// TIA Portal V15.1 export
// export: Created 2024-05-17T05:38:32.8666794Z, ExportSetting WithDefaults, DisplayName Totally Integrated Automation Portal, DisplayVersion V15.1 Update 5, DisplayName TIA Portal Openness, DisplayVersion V15.1 Update 5, DisplayName SINAMICS Startdrive Advanced, DisplayVersion V15.1, DisplayName G130, G150, S120, S150, SINAMICS MV, S210, DisplayVersion V15.1, DisplayName G110M, G120, G120C, G120D, G120P, DisplayVersion V15.1, DisplayName STEP 7 Professional, DisplayVersion V15.1 Update 5, DisplayName STEP 7 Safety, DisplayVersion V15.1, DisplayName WinCC Professional, DisplayVersion V15.1 Update 5, DisplayName SIMATIC Visualization Architect, DisplayVersion V15.1
FUNCTION_BLOCK "LAnInput2Lim"   // FB1707, FBD
TITLE = LAnInput2Lim
{ S7_Optimized_Access := 'FALSE' }
AUTHOR : VCC
FAMILY : ProcEqp
NAME : AnInput2
VERSION : 1.0
// ================================================================================
// This module is used to read an analogue Input value and scale it. 
// It also gives the possibility to define 2 limits (High and Low) and to create  
// alarms for these limits. 
// ================================================================================
// stored: AutoNumber false, IsIECCheckEnabled false, SetENOAutomatically False, UDAEnableTagReadback false
   VAR_INPUT
      I_AnInput { ExternalAccessible := 'False'; ExternalVisible := 'False'; ExternalWritable := 'False'} : Int;   // Analogue Input Value
      I_AnInput_Bipolar { ExternalAccessible := 'False'; ExternalVisible := 'False'; ExternalWritable := 'False'} : Bool;   // TRUE if Analogue Input Bipolar
      I_EnHAlarm { ExternalAccessible := 'False'; ExternalVisible := 'False'; ExternalWritable := 'False'} : Bool;   // Enable H Limit Alarm
      I_ResHAlarm { ExternalAccessible := 'False'; ExternalVisible := 'False'; ExternalWritable := 'False'} : Bool;   // Reset H Limit Alarm
      I_EnLAlarm { ExternalAccessible := 'False'; ExternalVisible := 'False'; ExternalWritable := 'False'} : Bool;   // Enable L Limit Alarm
      I_ResLAlarm { ExternalAccessible := 'False'; ExternalVisible := 'False'; ExternalWritable := 'False'} : Bool;   // Reset L Limit Alarm
      I_AlarmResetPB { ExternalAccessible := 'False'; ExternalVisible := 'False'; ExternalWritable := 'False'} : Bool;   // Alarm reset PB
   END_VAR
   VAR_OUTPUT
      O_SensorAlarm { ExternalAccessible := 'False'; ExternalVisible := 'False'; ExternalWritable := 'False'} : Bool;   // Sensor out of range
      O_HAlarm { ExternalAccessible := 'False'; ExternalVisible := 'False'; ExternalWritable := 'False'} : Bool;   // H Limit Alarm
      O_LAlarm { ExternalAccessible := 'False'; ExternalVisible := 'False'; ExternalWritable := 'False'} : Bool;   // L Limit Alarm
      O_AnInputScaled : Real;   // Analogue Input value after scaling
      O_AlarmABCondition { ExternalAccessible := 'False'; ExternalVisible := 'False'; ExternalWritable := 'False'} : Bool;   // Alarm AB condition
      O_HReached { ExternalAccessible := 'False'; ExternalVisible := 'False'; ExternalWritable := 'False'} : Bool;   // High Limit Reached
      O_LReached { ExternalAccessible := 'False'; ExternalVisible := 'False'; ExternalWritable := 'False'} : Bool;   // Low Limit Reached
      H_IAnim { ExternalAccessible := 'False'; ExternalVisible := 'False'; ExternalWritable := 'False'} : Word;   // HMI Animation of the icon
   END_VAR
   VAR DB_SPECIFIC
      H_In : Struct   // HMI
         AnInput_HighLimit : Real;   // From HMI : High Limit For Scaling Analogue Input
         AnInput_LowLimit : Real;   // From HMI : Low Limit For Scaling Analogue Input
         HHysteresis : Real;   // From HMI : Hysteresis value for High Limits
         LHysteresis : Real;   // From HMI : Hysteresis value for Low Limits
         HLimitValue : Real;   // From HMI : High Limit Value
         LLimitValue : Real;   // From HMI : Low Limit Value
         TimeDelay : DInt;   // From HMI : Time delay for limits
         Forcing : Bool;   // From HMI : True if forced value must be used
         ForcedAnInput : Real;   // From HMI : Forced Analogue Input Value
      END_STRUCT;
      H_Out : Struct   // HMI
         Anim : Word;   // HMI Animation of the object
         DBnr : Int;   // HMI Animation DB number
      END_STRUCT;
   END_VAR
   VAR
      HLimitTimer { ExternalAccessible := 'False'; ExternalVisible := 'False'; ExternalWritable := 'False'; S7_SetPoint := 'True'} : "LTimer";   // Timer H Limit
      LLimitTimer { ExternalAccessible := 'False'; ExternalVisible := 'False'; ExternalWritable := 'False'; S7_SetPoint := 'True'} : "LTimer";   // Timer L Limit
   END_VAR
   VAR DB_SPECIFIC
      AnInputScaled { ExternalAccessible := 'False'; ExternalVisible := 'False'; ExternalWritable := 'False'} : Real;   // Analogue Input value after scaling
      HTempSR { ExternalAccessible := 'False'; ExternalVisible := 'False'; ExternalWritable := 'False'} : Bool;   // Temp variable for SET/RESET
      LTempSR { ExternalAccessible := 'False'; ExternalVisible := 'False'; ExternalWritable := 'False'} : Bool;   // Temp variable for SET/RESET
      Scale_status { ExternalAccessible := 'False'; ExternalVisible := 'False'; ExternalWritable := 'False'} : Word;   // Status word for scaling operation
      HlimitHyst { ExternalAccessible := 'False'; ExternalVisible := 'False'; ExternalWritable := 'False'} : Real;   // H Limit with Hysteresis
      LlimitHyst { ExternalAccessible := 'False'; ExternalVisible := 'False'; ExternalWritable := 'False'} : Real;   // L Limit with Hysteresis
      HReached { ExternalAccessible := 'False'; ExternalVisible := 'False'; ExternalWritable := 'False'} : Bool;   // Temp variable H Limit Reached
      LReached { ExternalAccessible := 'False'; ExternalVisible := 'False'; ExternalWritable := 'False'} : Bool;   // Temp variable L Limit Reached
      HAlarmAlmCond { ExternalAccessible := 'False'; ExternalVisible := 'False'; ExternalWritable := 'False'} : Bool;   // HAlarm alarm condition
      LAlarmAlmCond { ExternalAccessible := 'False'; ExternalVisible := 'False'; ExternalWritable := 'False'} : Bool;   // LAlarm alarm condition
      HAlarm { ExternalAccessible := 'False'; ExternalVisible := 'False'; ExternalWritable := 'False'} : Bool;   // H Limit Alarm
      LAlarm { ExternalAccessible := 'False'; ExternalVisible := 'False'; ExternalWritable := 'False'} : Bool;   // L Limit Alarm
      SensorAlarm { ExternalAccessible := 'False'; ExternalVisible := 'False'; ExternalWritable := 'False'} : Bool;   // Sensor out of range
      SensorAlmCond { ExternalAccessible := 'False'; ExternalVisible := 'False'; ExternalWritable := 'False'} : Bool;   // Sensor alarm condition
      ScaleRetValue { ExternalAccessible := 'False'; ExternalVisible := 'False'; ExternalWritable := 'False'} : Int;   // Scale return value
      AnInputTmp { ExternalAccessible := 'False'; ExternalVisible := 'False'; ExternalWritable := 'False'} : Real;   // Analog input temporary
      DBnr { ExternalAccessible := 'False'; ExternalVisible := 'False'; ExternalWritable := 'False'} : Int;   // HMI DB number
   END_VAR
   VAR
      H_Alarm { ExternalAccessible := 'False'; ExternalVisible := 'False'; ExternalWritable := 'False'; S7_SetPoint := 'True'} : "LProc1AlarmMultiIn";
      L_Alarm { ExternalAccessible := 'False'; ExternalVisible := 'False'; ExternalWritable := 'False'; S7_SetPoint := 'True'} : "LProc1AlarmMultiIn";
      SensorAlm { ExternalAccessible := 'False'; ExternalVisible := 'False'; ExternalWritable := 'False'; S7_SetPoint := 'True'} : "LProc1AlarmMultiIn";
   END_VAR
BEGIN

NETWORK
TITLE = **** 1 - Inputs **** DB number
// DB number
      L     DINO;
      T     #DBnr;

REGION Network 2: **** 2.2 - Alarms - Alarm generation **** Alarm High Limit
   // Alarm High Limit
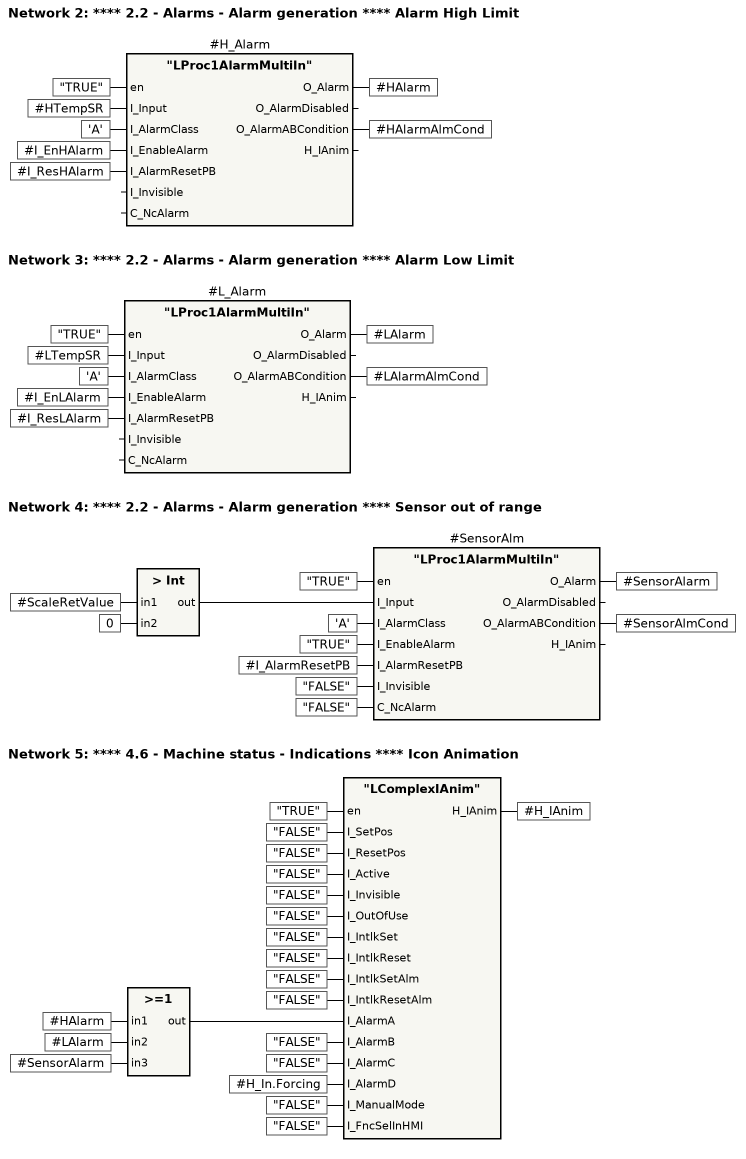
   IF "TRUE" THEN
       #H_Alarm(I_Input := #HTempSR,   // "LProc1AlarmMultiIn"
                I_AlarmClass := 'A',
                I_EnableAlarm := #I_EnHAlarm,
                I_AlarmResetPB := #I_ResHAlarm,
                O_Alarm => #HAlarm,
                O_AlarmABCondition => #HAlarmAlmCond);
   END_IF;
END_REGION

REGION Network 3: **** 2.2 - Alarms - Alarm generation **** Alarm Low Limit
   // Alarm Low Limit
   IF "TRUE" THEN
       #L_Alarm(I_Input := #LTempSR,   // "LProc1AlarmMultiIn"
                I_AlarmClass := 'A',
                I_EnableAlarm := #I_EnLAlarm,
                I_AlarmResetPB := #I_ResLAlarm,
                O_Alarm => #LAlarm,
                O_AlarmABCondition => #LAlarmAlmCond);
   END_IF;
END_REGION

REGION Network 4: **** 2.2 - Alarms - Alarm generation **** Sensor out of range
   // Sensor out of range
   IF "TRUE" THEN
       #SensorAlm(I_Input := #ScaleRetValue > 0,   // "LProc1AlarmMultiIn"
                  I_AlarmClass := 'A',
                  I_EnableAlarm := "TRUE",
                  I_AlarmResetPB := #I_AlarmResetPB,
                  I_Invisible := "FALSE",
                  C_NcAlarm := "FALSE",
                  O_Alarm => #SensorAlarm,
                  O_AlarmABCondition => #SensorAlmCond);
   END_IF;
END_REGION

REGION Network 5: **** 4.6 - Machine status - Indications **** Icon Animation
   // Icon Animation
   IF "TRUE" THEN
       "LComplexIAnim"(I_SetPos := "FALSE",
                       I_ResetPos := "FALSE",
                       I_Active := "FALSE",
                       I_Invisible := "FALSE",
                       I_OutOfUse := "FALSE",
                       I_IntlkSet := "FALSE",
                       I_IntlkReset := "FALSE",
                       I_IntlkSetAlm := "FALSE",
                       I_IntlkResetAlm := "FALSE",
                       I_AlarmA := #HAlarm OR #LAlarm OR #SensorAlarm,
                       I_AlarmB := "FALSE",
                       I_AlarmC := "FALSE",
                       I_AlarmD := #H_In.Forcing,
                       I_ManualMode := "FALSE",
                       I_FncSelInHMI := "FALSE",
                       H_IAnim => #H_IAnim);
   END_IF;
END_REGION

REGION Network 6: **** 4.6 - Machine status - Indications **** Animation
   // Animation
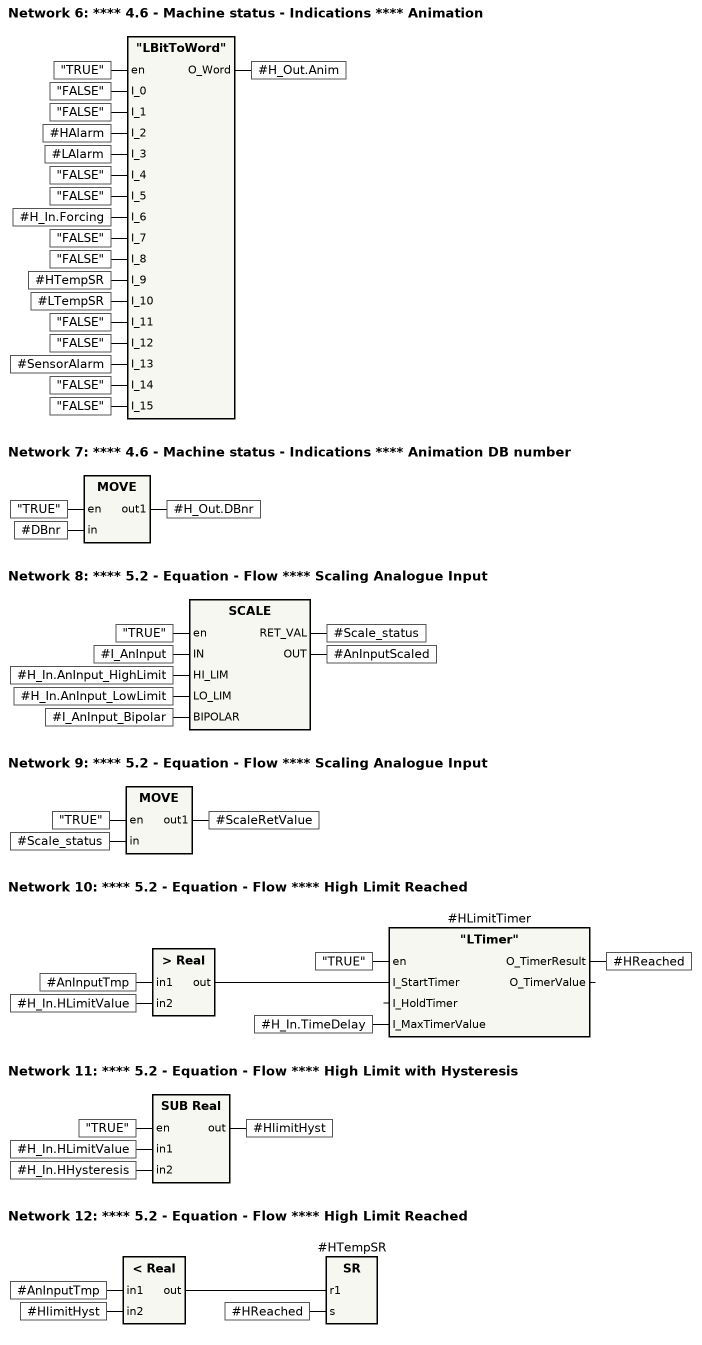
   IF "TRUE" THEN
       "LBitToWord"(I_0 := "FALSE",
                    I_1 := "FALSE",
                    I_2 := #HAlarm,
                    I_3 := #LAlarm,
                    I_4 := "FALSE",
                    I_5 := "FALSE",
                    I_6 := #H_In.Forcing,
                    I_7 := "FALSE",
                    I_8 := "FALSE",
                    I_9 := #HTempSR,
                    I_10 := #LTempSR,
                    I_11 := "FALSE",
                    I_12 := "FALSE",
                    I_13 := #SensorAlarm,
                    I_14 := "FALSE",
                    I_15 := "FALSE",
                    O_Word => #H_Out.Anim);
   END_IF;
END_REGION

REGION Network 7: **** 4.6 - Machine status - Indications **** Animation DB number
   // Animation DB number
   IF "TRUE" THEN #H_Out.DBnr := #DBnr; END_IF;
END_REGION

REGION Network 8: **** 5.2 - Equation - Flow **** Scaling Analogue Input
   // Scaling Analogue Input
   IF "TRUE" THEN
       #Scale_status := SCALE(IN := #I_AnInput,
                              HI_LIM := #H_In.AnInput_HighLimit,
                              LO_LIM := #H_In.AnInput_LowLimit,
                              BIPOLAR := #I_AnInput_Bipolar,
                              OUT => #AnInputScaled);
   END_IF;
END_REGION

REGION Network 9: **** 5.2 - Equation - Flow **** Scaling Analogue Input
   // Scaling Analogue Input
   IF "TRUE" THEN #ScaleRetValue := #Scale_status; END_IF;
END_REGION

REGION Network 10: **** 5.2 - Equation - Flow **** High Limit Reached
   // High Limit Reached
   IF "TRUE" THEN
       #HLimitTimer(I_StartTimer := #AnInputTmp > #H_In.HLimitValue,   // "LTimer"
                    I_MaxTimerValue := #H_In.TimeDelay,
                    O_TimerResult => #HReached);
   END_IF;
END_REGION

REGION Network 11: **** 5.2 - Equation - Flow **** High Limit with Hysteresis
   // High Limit with Hysteresis
   IF "TRUE" THEN #HlimitHyst := #H_In.HLimitValue - #H_In.HHysteresis; END_IF;
END_REGION

REGION Network 12: **** 5.2 - Equation - Flow **** High Limit Reached
   // High Limit Reached
   IF #HReached THEN
       #HTempSR := TRUE;   // SR flip-flop
   END_IF;
   IF #AnInputTmp < #HlimitHyst THEN #HTempSR := FALSE; END_IF;
END_REGION

REGION Network 13: **** 5.2 - Equation - Flow **** Low Limit Reached
   // Low Limit Reached
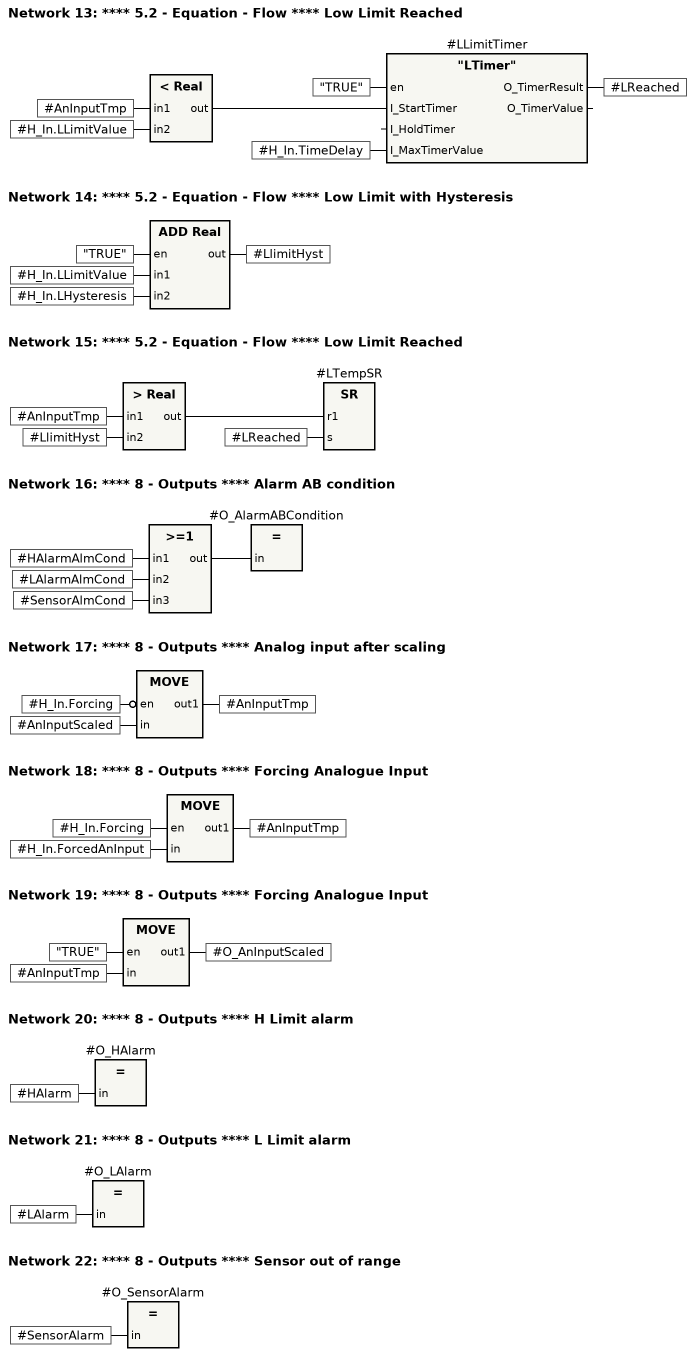
   IF "TRUE" THEN
       #LLimitTimer(I_StartTimer := #AnInputTmp < #H_In.LLimitValue,   // "LTimer"
                    I_MaxTimerValue := #H_In.TimeDelay,
                    O_TimerResult => #LReached);
   END_IF;
END_REGION

REGION Network 14: **** 5.2 - Equation - Flow **** Low Limit with Hysteresis
   // Low Limit with Hysteresis
   IF "TRUE" THEN #LlimitHyst := #H_In.LLimitValue + #H_In.LHysteresis; END_IF;
END_REGION

REGION Network 15: **** 5.2 - Equation - Flow **** Low Limit Reached
   // Low Limit Reached
   IF #LReached THEN
       #LTempSR := TRUE;   // SR flip-flop
   END_IF;
   IF #AnInputTmp > #LlimitHyst THEN #LTempSR := FALSE; END_IF;
END_REGION

REGION Network 16: **** 8 - Outputs **** Alarm AB condition
   // Alarm AB condition
   #O_AlarmABCondition := #HAlarmAlmCond OR #LAlarmAlmCond OR #SensorAlmCond;
END_REGION

REGION Network 17: **** 8 - Outputs **** Analog input after scaling
   // Analog input after scaling
   IF NOT #H_In.Forcing THEN #AnInputTmp := #AnInputScaled; END_IF;
END_REGION

REGION Network 18: **** 8 - Outputs **** Forcing Analogue Input
   // Forcing Analogue Input
   IF #H_In.Forcing THEN #AnInputTmp := #H_In.ForcedAnInput; END_IF;
END_REGION

REGION Network 19: **** 8 - Outputs **** Forcing Analogue Input
   // Forcing Analogue Input
   IF "TRUE" THEN #O_AnInputScaled := #AnInputTmp; END_IF;
END_REGION

REGION Network 20: **** 8 - Outputs **** H Limit alarm
   // H Limit alarm
   #O_HAlarm := #HAlarm;
END_REGION

REGION Network 21: **** 8 - Outputs **** L Limit alarm
   // L Limit alarm
   #O_LAlarm := #LAlarm;
END_REGION

REGION Network 22: **** 8 - Outputs **** Sensor out of range
   // Sensor out of range
   #O_SensorAlarm := #SensorAlarm;
END_REGION

REGION Network 23: **** 8 - Outputs **** H Limit reached
   // H Limit reached
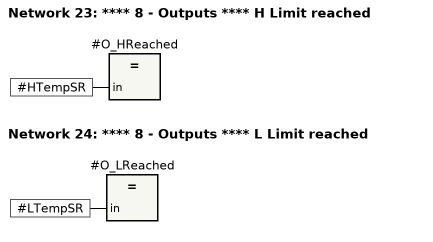
   #O_HReached := #HTempSR;
END_REGION

REGION Network 24: **** 8 - Outputs **** L Limit reached
   // L Limit reached
   #O_LReached := #LTempSR;
END_REGION
END_FUNCTION_BLOCK
